{attribute 'qualified_only'}
{attribute 'strict'}
{attribute 'to_string'}
TYPE E_AssemblyStationState :
(
    Disabled                    := 0,
    RecoveringSlideRetracted    := 10,
    RecoveringGripperOpen       := 20,
    RecoveringRotationPlace     := 30,

    Idle                        := 100,
    ExtendingSlideToPick        := 110,
    DelayAfterPickExtend        := 120,
    ClosingGripper              := 130,
    DelayAfterGripperClose      := 140,
    RetractingSlideWithPart     := 150,
    DelayAfterPickRetract       := 160,

    RotatingToPlace             := 170,
    DelayAfterRotateToPlace     := 180,

    ExtendingSlideToPlace       := 190,
    DelayAfterPlaceExtend       := 200,

    OpeningGripper              := 210,
    DelayAfterGripperOpen       := 220,

    RetractingSlideHome         := 230,
    DelayAfterHomeRetract       := 240,

    RotatingToPick              := 250,
    DelayAfterRotateToPick      := 260,

    Complete                    := 270,

    Fault                       := 999
);
END_TYPE

(* stored: Version 1.1.0.1, ProductVersion 3.1.4026.18
   DUT E_AssemblyStationState: Id {625786e8-f610-403e-8b03-95f9cd71c417} *)
